(* CoDeSys 2.3.9.31 project: TEST2017051301.pro *)
(* Libraries: STANDARD.LIB 5.6.98 11:03:02 *)

(* Task configuration *)
TASK Standard (PRIORITY := 0, INTERVAL := T#10ms);
	Left_Feed();
	Left_Move();
	Cycle_1();
END_TASK

(* Global variable list: Global_Variables *)
VAR_GLOBAL
	M0 :BOOL;
	M1: BOOL;
END_VAR

(* POU Left_Feed, ST *)
PROGRAM Left_Feed
VAR
	A1: BOOL;
END_VAR
A1 := M1;
END_PROGRAM

(* POU Left_Move, ST *)
PROGRAM Left_Move
VAR
	B2: BOOL;
END_VAR
B2 := M1;
END_PROGRAM

(* POU Cycle_1, LD *)
PROGRAM Cycle_1
VAR
	T1: TON;

	T2: TON;
END_VAR
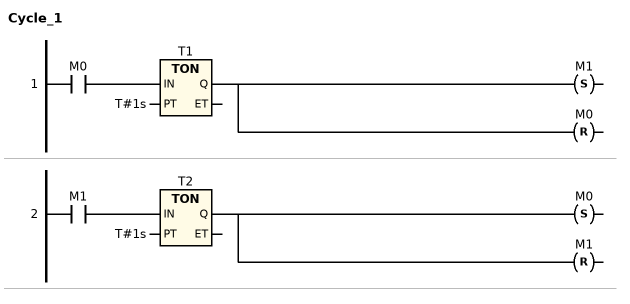
_LD_ (* Ladder Diagram *)
NETWORK 1
	[M0] - T1:TON(IN: *, PT: T#1s) --- (S M1) (R M0)
NETWORK 2
	[M1] - T2:TON(IN: *, PT: T#1s) --- (S M0) (R M1)
_END_LD_
(* the same logic as Structured Text *)
(* Network 1 *)
T1(IN := M0, PT := T#1s);
IF T1.Q THEN M1 := TRUE; M0 := FALSE; END_IF;
(* Network 2 *)
T2(IN := M1, PT := T#1s);
IF T2.Q THEN M0 := TRUE; M1 := FALSE; END_IF;
END_PROGRAM
